FUNCTION_BLOCK public FB_AbstractLoggerFactory
VAR_INPUT
END_VAR
VAR_OUTPUT
END_VAR
VAR
END_VAR

METHOD PUBLIC GetLogger : ILogger
VAR_INPUT
END_VAR
;
END_METHOD

END_FUNCTION_BLOCK

(* stored: Version 1.1.0.1, ProductVersion 3.1.0.24
   POU FB_AbstractLoggerFactory: Id {03cfff1e-2141-489d-a35f-4c2a1a94d4d9}
   Method GetLogger: Id {36432c5d-7b99-47b1-85f8-5ffc6a59e86f} *)
